GLOBALCONSTANTS storageStatusMessages (* Global constants *)
  (* Standard: 61499-1 *)
  (* Version 1.0, 2026-06-13, franz *)
  PACKAGE logiBUS::storage::const;
  VAR_GLOBAL CONSTANT
    OK : STRING := 'OK';
    NOOP : STRING := 'Value was not stored. Old is new';
  END_VAR
END_GLOBALCONSTANTS
